{attribute addProperty BoxType "KL3351"}
{attribute addProperty Id "Channel_1Channel_274E4E9000"}
{attribute addProperty CRC "2203132032"}
{attribute addProperty SizeInBites "0"}
{attribute addProperty SizeInBytes "0"}
TYPE KL3351_83512080 :
STRUCT
	{attribute addProperty Name "Channel_1"}
	Channel_1 : Channel_274E4E90;
END_STRUCT
END_TYPE

(* stored: Version 1.2.0.0, ProductVersion 3.1.4024.9
   DUT KL3351_83512080: Id {22b20d1d-c79c-461d-8ee6-b0ea7f51de3e} *)
